///Data reciever interface, implement this interface in the block
///that has to recieve data 
INTERFACE IDataReciever

// New data recieved
METHOD NewDataRecieved : HResult
VAR_INPUT
    data : Data; ///Data recieved
END_VAR
END_METHOD

END_INTERFACE

(* stored: Version 1.1.0.1, ProductVersion 3.1.4020.12
   Itf IDataReciever: Id {2443fb2b-c3a2-4e64-98e5-c23932d17bef}
   Method NewDataRecieved: Id {b7ee0f63-4c37-40c8-b765-f1d990907cc5} *)
